(* Schneider Machine Expert - Basic project Redundant_Motors_v3, file version 3.0.0.0 *)
(* ProjectInformations: Name=New project *)

HARDWARE
  Cpu 0: TM221CE16T
  EthernetConfiguration: NetworkName=M221, IpAllocationMode=FixedAddress, IpAddress=0.0.0.0, SubnetMask=0.0.0.0
  SerialLineConfiguration: Baud=Baud19200, Parity=ParityEven, DataBits=DataBits8, StopBits=StopBits1, PhysicalMedium=PhysicalMediumRs485, TransmissionMode=TransmissionModeModbusRtu, SlaveId=1, Addressing=SlaveAddressing
  MastTask: UsePeriodScanMode=false, PeriodScan=100
  FastTask: Period=255
  CpuBehavior: StartingMode=StartAsPreviousState, AutoSaveRamOnEeprom=true, WatchdogPeriod=250

SYMBOLS  (address, symbol, comment, settings)
  %M0       SYSTEM_READY  "System ready after 3s startup"
  %M1       RUN_REQUEST  "Operator run request"
  %M2       M1_CMD  "Motor 1 command"
  %M3       M2_CMD  "Motor 2 command"
  %M4       M1_RUNNING  "Motor 1 running feedback"
  %M5       M2_RUNNING  "Motor 2 running feedback"
  %M6       M1_FAIL  "Motor 1 failure alarm"
  %M7       M2_FAIL  "Motor 2 failure alarm"
  %M8       M1_OL_ALARM  "Motor 1 overload alarm"
  %M9       M2_OL_ALARM  "Motor 2 overload alarm"
  %S0       SB_COLDSTART  "Indicates or executes a cold start (data initialized to default values)"
  %S1       SB_WARMSTART  "Indicates there was a warm start with data backup"
  %TM0      STARTUP_TMR  "System startup delay"  [Preset=3, Base=OneSecond]
  %TM1      M1_START_TMR  "M1 startup timeout"  [Preset=5, Base=OneSecond]
  %TM2      M2_START_TMR  "M2 startup timeout"  [Preset=5, Base=OneSecond]
  %I0.0     EMERGENCY_PB

POU New POU
  (* SectionNumber=0 *)

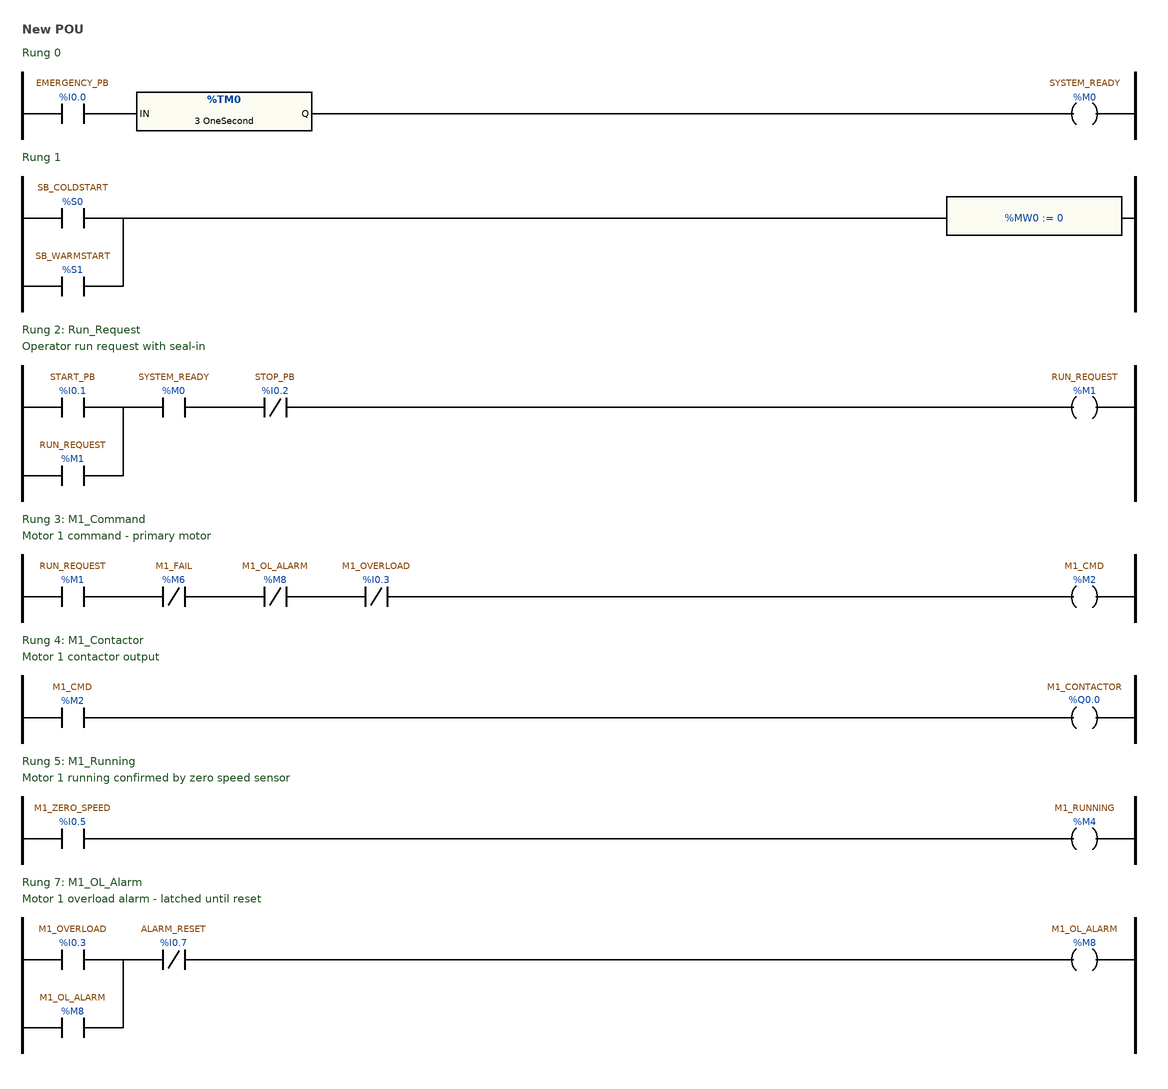

// Rung 0
  BLK %TM0                (* STARTUP_TMR *)
  LD %I0.0                (* EMERGENCY_PB *)
  IN
  OUT_BLK
  LD Q
  ST %M0                  (* SYSTEM_READY *)
  END_BLK
  // as ST:
  //   STARTUP_TMR(IN := EMERGENCY_PB);
  //   SYSTEM_READY := STARTUP_TMR.Q;

// Rung 1
  LD %S0                  (* SB_COLDSTART *)
  OR %S1                  (* SB_WARMSTART *)
  [ %MW0 := 0 ]
  // as ST:
  //   IF SB_COLDSTART OR SB_WARMSTART THEN %MW0 := 0; END_IF;

// Rung 2: Run_Request
// Operator run request with seal-in
  LD %I0.1
  OR %M1                  (* RUN_REQUEST *)
  AND %M0                 (* SYSTEM_READY *)
  ANDN %I0.2
  ST %M1                  (* RUN_REQUEST *)
  // %I0.1: Start Button
  // %M0: System Ready
  // %I0.2: Stop NC
  // %M1: Run Request
  // %M1: Seal-in
  // as ST:
  //   RUN_REQUEST := (%I0.1 OR RUN_REQUEST) AND SYSTEM_READY AND NOT %I0.2;

// Rung 3: M1_Command
// Motor 1 command - primary motor
  LD %M1                  (* RUN_REQUEST *)
  ANDN %M6                (* M1_FAIL *)
  ANDN %M8                (* M1_OL_ALARM *)
  ANDN %I0.3
  ST %M2                  (* M1_CMD *)
  // %M1: Run Req
  // %M6: M1 OK
  // %M8: No OL
  // %I0.3: OL OK
  // %M2: M1 Cmd
  // as ST:
  //   M1_CMD := RUN_REQUEST AND NOT M1_FAIL AND NOT M1_OL_ALARM AND NOT %I0.3;

// Rung 4: M1_Contactor
// Motor 1 contactor output
  LD %M2                  (* M1_CMD *)
  ST %Q0.0
  // %M2: M1 Cmd
  // %Q0.0: M1 Cont
  // as ST:
  //   %Q0.0 := M1_CMD;

// Rung 5: M1_Running
// Motor 1 running confirmed by zero speed sensor
  LD %I0.5
  ST %M4                  (* M1_RUNNING *)
  // %I0.5: M1 Speed
  // %M4: M1 Run
  // as ST:
  //   M1_RUNNING := %I0.5;

// Rung 6: M1_Fail
// Motor 1 failure alarm - latched until reset
  LD %M2                  (* M1_CMD *)
  ANDN %M4                (* M1_RUNNING *)
  AND %TM1.Q              (* M1_START_TMR *)
  OR %M6                  (* M1_FAIL *)
  ANDN %I0.7
  ST %M6                  (* M1_FAIL *)
  // %M2: M1 Cmd
  // %M4: Not Run
  // %TM1.Q: 5s Done
  // %I0.7: No Reset
  // %M6: M1 Fail
  // %M6: Latch
  // as ST:
  //   M1_FAIL := (M1_CMD AND NOT M1_RUNNING AND M1_START_TMR.Q OR M1_FAIL) AND NOT %I0.7;
  (* the ladder stored for this rung does not match its IL; not drawn *)

// Rung 7: M1_OL_Alarm
// Motor 1 overload alarm - latched until reset
  LD %I0.3
  OR %M8                  (* M1_OL_ALARM *)
  ANDN %I0.7
  ST %M8                  (* M1_OL_ALARM *)
  // %I0.3: M1 OL
  // %I0.7: No Reset
  // %M8: M1 OL Alm
  // %M8: Latch
  // as ST:
  //   M1_OL_ALARM := (%I0.3 OR M1_OL_ALARM) AND NOT %I0.7;

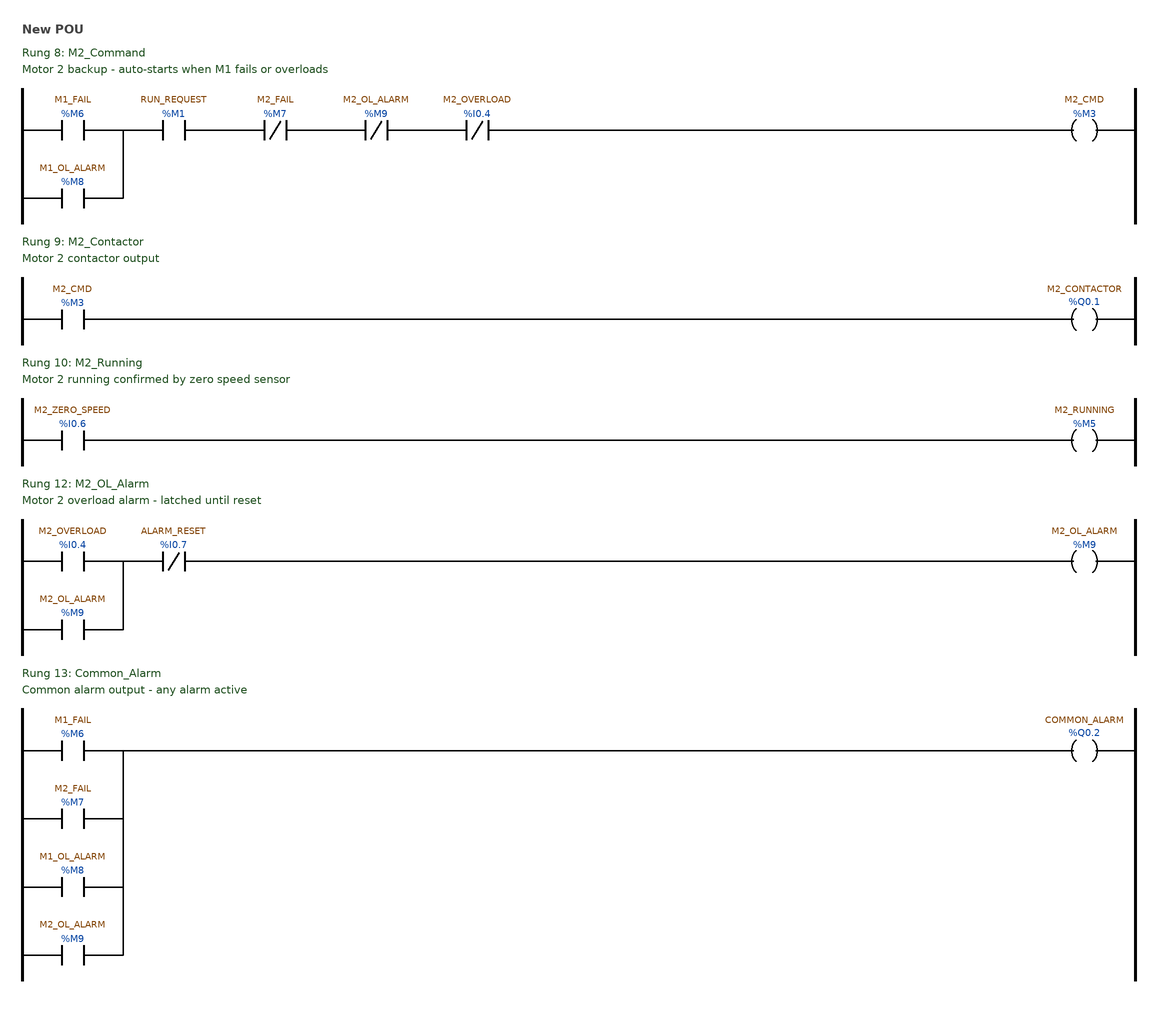

// Rung 8: M2_Command
// Motor 2 backup - auto-starts when M1 fails or overloads
  LD %M6                  (* M1_FAIL *)
  OR %M8                  (* M1_OL_ALARM *)
  AND %M1                 (* RUN_REQUEST *)
  ANDN %M7                (* M2_FAIL *)
  ANDN %M9                (* M2_OL_ALARM *)
  ANDN %I0.4
  ST %M3                  (* M2_CMD *)
  // %M6: M1 Fail
  // %M1: Run Req
  // %M7: M2 OK
  // %M9: No M2 OL
  // %I0.4: M2 OL OK
  // %M3: M2 Cmd
  // %M8: M1 OL
  // as ST:
  //   M2_CMD := (M1_FAIL OR M1_OL_ALARM) AND RUN_REQUEST AND NOT M2_FAIL AND NOT M2_OL_ALARM AND NOT %I0.4;

// Rung 9: M2_Contactor
// Motor 2 contactor output
  LD %M3                  (* M2_CMD *)
  ST %Q0.1
  // %M3: M2 Cmd
  // %Q0.1: M2 Cont
  // as ST:
  //   %Q0.1 := M2_CMD;

// Rung 10: M2_Running
// Motor 2 running confirmed by zero speed sensor
  LD %I0.6
  ST %M5                  (* M2_RUNNING *)
  // %I0.6: M2 Speed
  // %M5: M2 Run
  // as ST:
  //   M2_RUNNING := %I0.6;

// Rung 11: M2_Fail
// Motor 2 failure alarm - latched until reset
  LD %M3                  (* M2_CMD *)
  ANDN %M5                (* M2_RUNNING *)
  AND %TM2.Q              (* M2_START_TMR *)
  OR %M7                  (* M2_FAIL *)
  ANDN %I0.7
  ST %M7                  (* M2_FAIL *)
  // %M3: M2 Cmd
  // %M5: Not Run
  // %TM2.Q: 5s Done
  // %I0.7: No Reset
  // %M7: M2 Fail
  // %M7: Latch
  // as ST:
  //   M2_FAIL := (M2_CMD AND NOT M2_RUNNING AND M2_START_TMR.Q OR M2_FAIL) AND NOT %I0.7;
  (* the ladder stored for this rung does not match its IL; not drawn *)

// Rung 12: M2_OL_Alarm
// Motor 2 overload alarm - latched until reset
  LD %I0.4
  OR %M9                  (* M2_OL_ALARM *)
  ANDN %I0.7
  ST %M9                  (* M2_OL_ALARM *)
  // %I0.4: M2 OL
  // %I0.7: No Reset
  // %M9: M2 OL Alm
  // %M9: Latch
  // as ST:
  //   M2_OL_ALARM := (%I0.4 OR M2_OL_ALARM) AND NOT %I0.7;

// Rung 13: Common_Alarm
// Common alarm output - any alarm active
  LD %M6                  (* M1_FAIL *)
  OR %M7                  (* M2_FAIL *)
  OR %M8                  (* M1_OL_ALARM *)
  OR %M9                  (* M2_OL_ALARM *)
  ST %Q0.2
  // %M6: M1 Fail
  // %Q0.2: Alarm
  // %M7: M2 Fail
  // %M8: M1 OL
  // %M9: M2 OL
  // as ST:
  //   %Q0.2 := M1_FAIL OR M2_FAIL OR M1_OL_ALARM OR M2_OL_ALARM;
